KUKA KRL data list: Mill_LeafGlue.dat

&ACCESS RVEO
&REL 14
&PARAM EDITMASK = *
&PARAM TEMPLATE = C:\KRC\Roboter\Template\vorgabe
&PARAM DISKPATH = KRC:\R1\Program\LeafProfiles
DEFDAT Mill_LeafGlue

   ;Amount of glue holes
   DECL CONST INT iHoleSize = 4

   ;Gluehole profile edge offsetX
   DECL CONST REAL rGlueHoleOffsetX = 11.0

   ;Gluehole profile edge offsetY
   DECL CONST REAL rGlueHoleY[2]
   rGlueHoleY[1] = 13.0
   rGlueHoleY[2] = 67.5

ENDDAT
